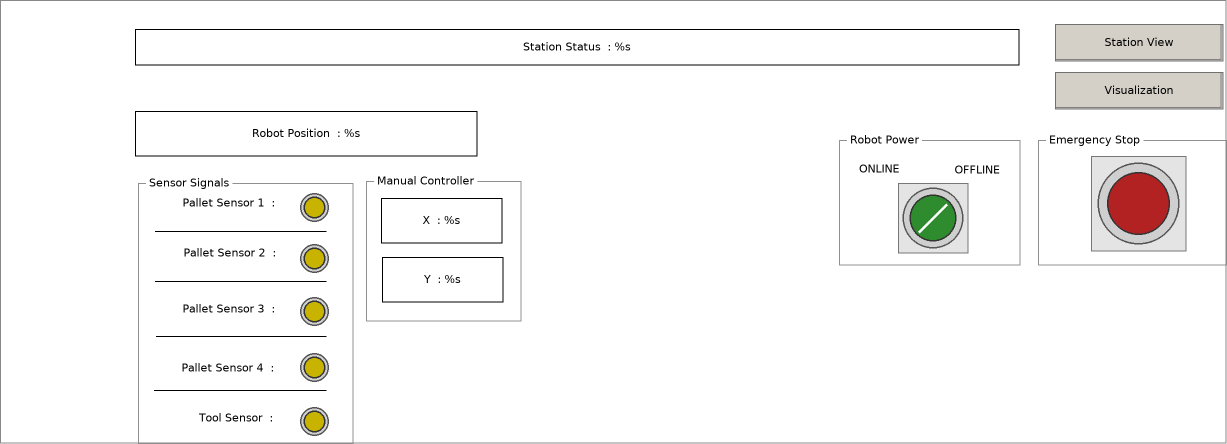
VISUALIZATION RobotStation  // 1227x444
    Rectangle (135,29 884x36), "Station Status : %s", text variable: Visualaisation_Control.mxStationStatus
    GroupBox (839,132 181x133), "Robot Power", invisible if: CommData.mxOnlineMode
        RotarySwitch (59,51 70x70), variable: CommData.mxRobotOnline, invisible if: CommData.mxOnlineMode, behaviour: TOGGLE, style: Switch-RotarySwitch-Green
        Label (11,22 59x30), "ONLINE"
        Label (106,23 65x30), "OFFLINE"
    Button (1055,72 168x37), "Visualization"
        OnMouseClick: change screen: Visualization
    GroupBox (1038,132 189x133), "Emergency Stop"
        PushSwitch (45,24 111x95), variable: GVL.ixEmergencyStop, behaviour: TOGGLE, style: Switch-PushSwitch-Red
    Rectangle (135,111 342x45), "Robot Position : %s", text variable: CommData.msRobotLastPos
    GroupBox (138,175 215x269), "Sensor Signals"
        Label (15,178 150x30), "Pallet Sensor 4 :"
        Label (17,63 150x30), "Pallet Sensor 2 :"
        Line (17,56) (188,56)
        Lamp1 (160,16 33x33), variable: GVL.ixInductiveSensor1, style: Lamp-Lamp1-Yellow
        Lamp1 (160,67 33x33), variable: GVL.ixInductiveSensor2, style: Lamp-Lamp1-Yellow
        Lamp1 (160,120 33x33), variable: GVL.ixInductiveSensor3, style: Lamp-Lamp1-Yellow
        Lamp1 (160,176 33x33), variable: GVL.ixInductiveSensor4, style: Lamp-Lamp1-Yellow
        Label (16,119 150x30), "Pallet Sensor 3 :"
        Label (23,228 150x30), "Tool Sensor :"
        Lamp1 (160,230 33x33), variable: GVL.ixInductiveSensorinTool, style: Lamp-Lamp1-Yellow
        Line (17,106) (188,106)
        Line (18,161) (188,161)
        Line (16,215) (188,215)
        Label (16,13 150x30), "Pallet Sensor 1 :"
    GroupBox (366,173 155x148), "Manual Controller"
        Rectangle (16,84 121x45), "Y : %s", text variable: CommData.mwYaxis
            OnMouseClick: write the text variable via Default
        Rectangle (15,25 121x45), "X : %s", text variable: CommData.mwXaxis
            OnMouseClick: write the text variable via Default
    Button (1055,24 168x37), "Station View"
        OnMouseClick: change screen: Station
END_VISUALIZATION

(* stored: Version 1.1.0.1, ProductVersion 3.1.4024.12
   Visu RobotStation: Id {d0399a33-d6a0-44fd-91ac-ef1763637ad4} *)
